// Mitsubishi GX Works2 project: Ex04   PLC: Q03UD

PROGRAM Lane1
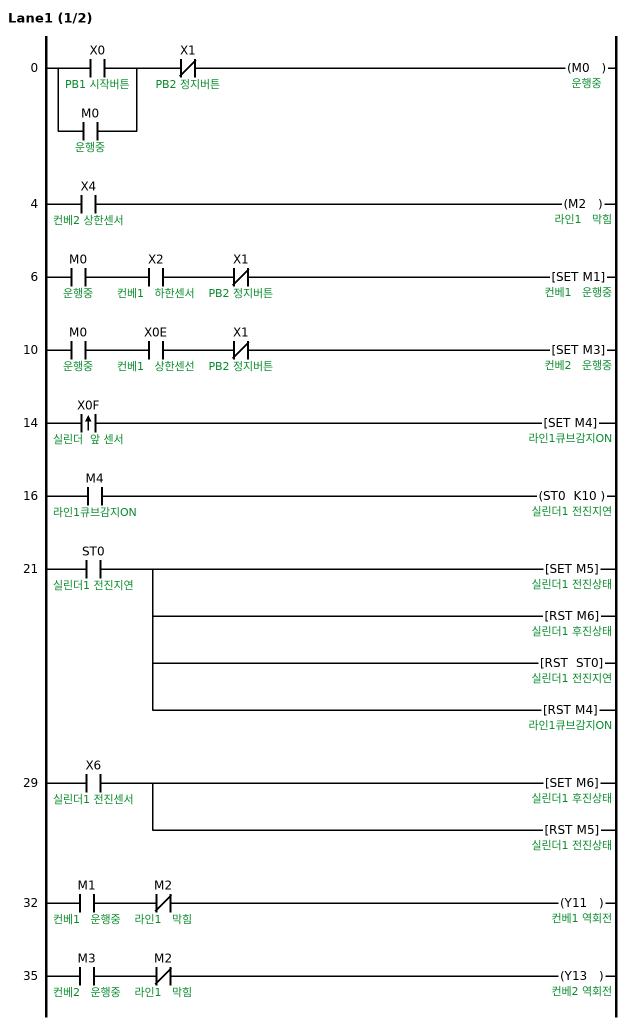
0     LD      X0  ; PB1 시작버튼
      OR      M0  ; 운행중
      ANI     X1  ; PB2 정지버튼
      OUT     M0  ; 운행중
4     LD      X4  ; 컨베2 상한센서
      OUT     M2  ; 라인1   막힘
6     LD      M0  ; 운행중
      AND     X2  ; 컨베1   하한센서
      ANI     X1  ; PB2 정지버튼
      SET     M1  ; 컨베1   운행중
10    LD      M0  ; 운행중
      AND     X0E  ; 컨베1   상한센선
      ANI     X1  ; PB2 정지버튼
      SET     M3  ; 컨베2   운행중
14    LDP     X0F  ; 실린더  앞 센서
      SET     M4  ; 라인1큐브감지ON
16    LD      M4  ; 라인1큐브감지ON
      OUT     ST0 K10  ; 실린더1 전진지연
21    LD      ST0  ; 실린더1 전진지연
      SET     M5  ; 실린더1 전진상태
      RST     M6  ; 실린더1 후진상태
      RST     ST0  ; 실린더1 전진지연
      RST     M4  ; 라인1큐브감지ON
29    LD      X6  ; 실린더1 전진센서
      SET     M6  ; 실린더1 후진상태
      RST     M5  ; 실린더1 전진상태
32    LD      M1  ; 컨베1   운행중
      ANI     M2  ; 라인1   막힘
      OUT     Y11  ; 컨베1 역회전
35    LD      M3  ; 컨베2   운행중
      ANI     M2  ; 라인1   막힘
      OUT     Y13  ; 컨베2 역회전
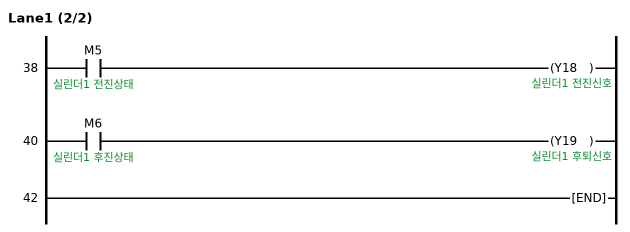
38    LD      M5  ; 실린더1 전진상태
      OUT     Y18  ; 실린더1 전진신호
40    LD      M6  ; 실린더1 후진상태
      OUT     Y19  ; 실린더1 후퇴신호
42    END
END_PROGRAM

PROGRAM Lane2
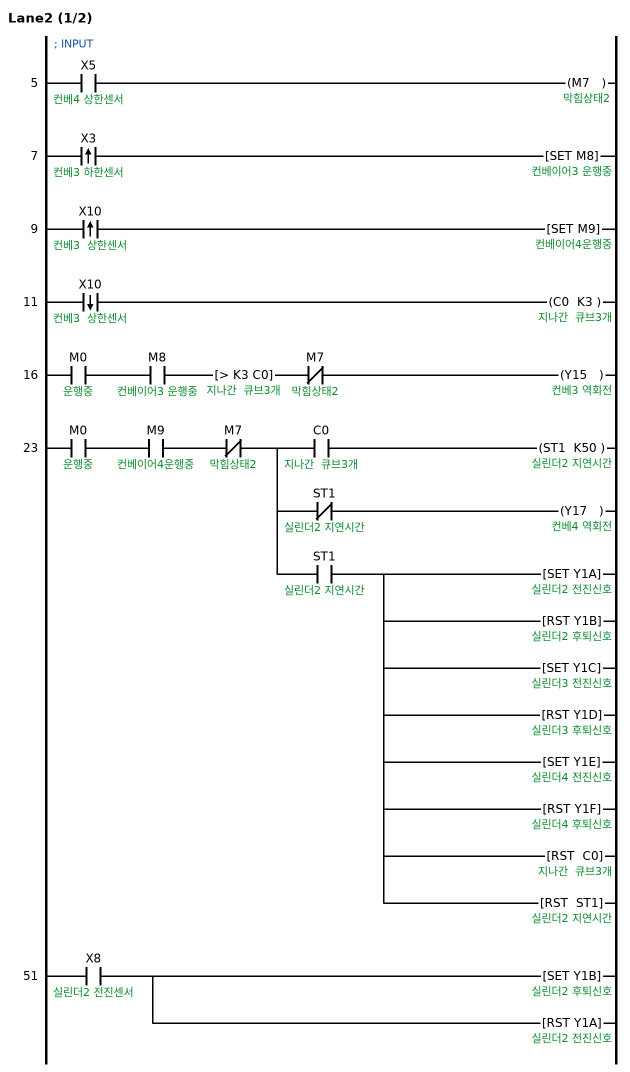
; INPUT
5     LD      X5  ; 컨베4 상한센서
      OUT     M7  ; 막힘상태2
7     LDP     X3  ; 컨베3 하한센서
      SET     M8  ; 컨베이어3 운행중
9     LDP     X10  ; 컨베3  상한센서
      SET     M9  ; 컨베이어4운행중
11    LDF     X10  ; 컨베3  상한센서
      OUT     C0 K3  ; 지나간  큐브3개
16    LD      M0  ; 운행중
      AND     M8  ; 컨베이어3 운행중
      AND>    K3 C0  ; 지나간  큐브3개
      ANI     M7  ; 막힘상태2
      OUT     Y15  ; 컨베3 역회전
23    LD      M0  ; 운행중
      AND     M9  ; 컨베이어4운행중
      ANI     M7  ; 막힘상태2
      MPS
      AND     C0  ; 지나간  큐브3개
      OUT     ST1 K50  ; 실린더2 지연시간
      MRD
      ANI     ST1  ; 실린더2 지연시간
      OUT     Y17  ; 컨베4 역회전
      MPP
      AND     ST1  ; 실린더2 지연시간
      SET     Y1A  ; 실린더2 전진신호
      RST     Y1B  ; 실린더2 후퇴신호
      SET     Y1C  ; 실린더3 전진신호
      RST     Y1D  ; 실린더3 후퇴신호
      SET     Y1E  ; 실린더4 전진신호
      RST     Y1F  ; 실린더4 후퇴신호
      RST     C0  ; 지나간  큐브3개
      RST     ST1  ; 실린더2 지연시간
51    LD      X8  ; 실린더2 전진센서
      SET     Y1B  ; 실린더2 후퇴신호
      RST     Y1A  ; 실린더2 전진신호
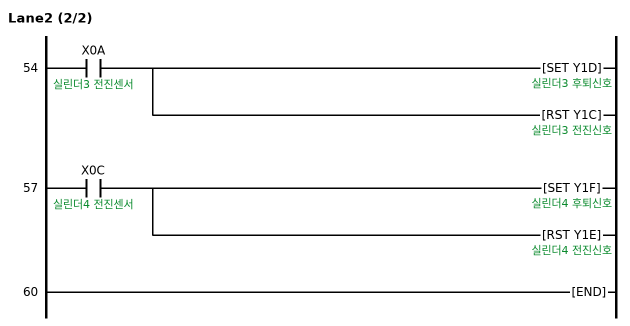
54    LD      X0A  ; 실린더3 전진센서
      SET     Y1D  ; 실린더3 후퇴신호
      RST     Y1C  ; 실린더3 전진신호
57    LD      X0C  ; 실린더4 전진센서
      SET     Y1F  ; 실린더4 후퇴신호
      RST     Y1E  ; 실린더4 전진신호
60    END
END_PROGRAM

// device comments not shown above
X7  ; 실린더1 후진센서
X9  ; 실린더2 후진센서
X0B  ; 실린더3 후진센서
X0D  ; 실린더4 후진센서
X11  ; 컨베3   하한센서
Y10  ; 컨베1 정회전
Y12  ; 컨베2 정회전
Y14  ; 컨베3 정회전
Y16  ; 컨베4 정회전
